{attribute 'GeneratedUsingTerminal: KL2535-0001'}
{attribute addProperty BoxType "KL2535-0001"}
{attribute addProperty Id "Channel_1AT %I*0Channel_2AT %I*0"}
{attribute addProperty CRC "1343494386"}
{attribute addProperty Size "0"}
TYPE KL_501418F2 :
STRUCT
	{attribute addProperty Name "Channel_1"}
	Channel_1 : ;
	{attribute addProperty Name "Channel_2"}
	Channel_2 : ;
END_STRUCT
END_TYPE

(* stored: Version 1.2.0.0, ProductVersion 3.1.4024.9
   DUT KL_501418F2: Id {1a0c1e3d-6f2b-4e48-afe2-b066263b5db4} *)
